INTERFACE I_XP_Trigger  EXTENDS __SYSTEM.IQueryInterface

{attribute 'monitoring':='call'}
PROPERTY AccocietedTrack : I_XP_Track
GET
END_GET
SET
END_SET
END_PROPERTY

{attribute 'monitoring':='call'}
PROPERTY HR : HRESULT
GET
END_GET
END_PROPERTY

PROPERTY ListOfMoversToCheck : I_CH_List
SET
END_SET
END_PROPERTY

{attribute 'monitoring':='call'}
PROPERTY MoverAtTrigger : I_XP_Mover
GET
END_GET
END_PROPERTY

{attribute 'monitoring':='call'}
PROPERTY MoverDetected : BOOL
GET
END_GET
END_PROPERTY

{attribute 'monitoring':='call'}
PROPERTY PositionOnTrack : LREAL
GET
END_GET
SET
END_SET
END_PROPERTY

{attribute 'monitoring':='call'}
PROPERTY TimeStamp : T_DCTIME64;
GET
END_GET
END_PROPERTY

{attribute 'monitoring':='call'}
PROPERTY TriggerDirection : Tc3_Mc3Definitions.MC_Direction
GET
END_GET
SET
END_SET
END_PROPERTY

END_INTERFACE

(* stored: Version 1.1.0.1, ProductVersion 3.1.4024.12
   Itf I_XP_Trigger: Id {e889dd59-5dee-4e00-b90b-22cc52226e89}
   Property AccocietedTrack: Id {ef546e42-ba12-4853-b3cc-e3135efdb3a0}
   Get Get: Id {b434b88a-019b-4891-8eb4-ce9ebdf862e3}
   Set Set: Id {f7b7a5fe-b6e6-4b19-9e92-2b4b10d34513}
   Property HR: Id {06d44635-3899-4ea3-949a-de9d327c067f}
   Get Get: Id {39fe9785-6fbf-4da0-a19c-335771fa6e58}
   Property ListOfMoversToCheck: Id {42534cb0-9df8-4806-972f-2059bafdf42f}
   Set Set: Id {f2d3cab5-804f-448e-96b1-3f5fdc6303b0}
   Property MoverAtTrigger: Id {fd27ac87-7291-46e9-88bc-eeae84dfef00}
   Get Get: Id {84e37e84-fd84-4616-b3d6-21ff5c4d115a}
   Property MoverDetected: Id {f3e18a86-2212-4fc8-8459-68b23c5ff674}
   Get Get: Id {2fbc8824-c313-4d36-b789-b3fb118d82cc}
   Property PositionOnTrack: Id {362a2ebc-f473-4db3-8f3e-aea905d1b2e1}
   Get Get: Id {eb74a73a-f59b-432c-becf-664cb07b2b77}
   Set Set: Id {83cdd31a-0ea3-4417-b1a4-e389b539f4f6}
   Property TimeStamp: Id {f5da10b0-5c07-47b8-b4d1-c81ce3f3f9d1}
   Get Get: Id {d4bad2b0-8d75-46b2-8133-7526ba2775de}
   Property TriggerDirection: Id {2e609c80-0dec-4a1b-9830-c24df066d715}
   Get Get: Id {2199bc2e-b8a3-4b8b-8bca-a38ea00b093e}
   Set Set: Id {935f9921-c87a-45b6-a856-7277def4e98e} *)
